{attribute addProperty BoxType "EL6201-0000-0017"}
{attribute addProperty Id "Slave_24A_DI0BIT10.125185Slave_24A_DI1BIT10.125186Slave_24A_DI2BIT10.125187Slave_24A_DI3BIT10.125188Slave_24B_DI0BIT10.125189Slave_24B_DI1BIT10.125190Slave_24B_DI2BIT10.125191Slave_24B_DI3BIT10.125192"}
{attribute addProperty CRC "3003379435"}
{attribute addProperty SizeInBites "8"}
{attribute addProperty SizeInBytes "1"}
TYPE Slave_24_Inputs_B303EEEB :
STRUCT
	{attribute addProperty Name "Slave_24A_DI0"}
	Slave_24A_DI0 : BIT;
	{attribute addProperty Name "Slave_24A_DI1"}
	Slave_24A_DI1 : BIT;
	{attribute addProperty Name "Slave_24A_DI2"}
	Slave_24A_DI2 : BIT;
	{attribute addProperty Name "Slave_24A_DI3"}
	Slave_24A_DI3 : BIT;
	{attribute addProperty Name "Slave_24B_DI0"}
	Slave_24B_DI0 : BIT;
	{attribute addProperty Name "Slave_24B_DI1"}
	Slave_24B_DI1 : BIT;
	{attribute addProperty Name "Slave_24B_DI2"}
	Slave_24B_DI2 : BIT;
	{attribute addProperty Name "Slave_24B_DI3"}
	Slave_24B_DI3 : BIT;
END_STRUCT
END_TYPE

(* stored: Version 1.2.0.0, ProductVersion 3.1.4024.9
   DUT Slave_24_Inputs_B303EEEB: Id {0cc37f9a-ec4c-44ef-bf4c-d32f27909fbb} *)
